KUKA KRL program: gestion_camara.src, gestion_camara.dat

--- gestion_camara.src ---
&ACCESS RVO2
&REL 8
&PARAM EDITMASK = *
&PARAM TEMPLATE = C:\KRC\Roboter\Template\vorgabe
DEF gestion_camara( )


END
GLOBAL DEF CAM_INI()

INPICKER_Handler.DataToSend.command=0
INPICKER_Handler.DataToSend.CameraID=0
INPICKER_Handler.DataToSend.ContainerID=0
INPICKER_Handler.DataToSend.GraspConfirmation=0
INPICKER_Handler.datatosend.partid=0

END
GLOBAL DEF CAM_CALIB_INI()

INPICKER_Handler.DataToSend.command=0
INPICKER_Handler.DataToSend.CameraID=1
INPICKER_Handler.DataToSend.ContainerID=0
INPICKER_Handler.DataToSend.GraspConfirmation=0
INPICKER_Handler.datatosend.partid=1

END

GLOBAL DEF CAM_CALIB_FOTO(P_IN :IN)
INT P_IN

INPICKER_Handler.DataToSend.command=0
wait for (INPICKER_Handler.DataReceived.state==0)
INPICKER_Handler.DataToSend.GraspConfirmation=P_IN
INPICKER_Handler.DataToSend.command=3
wait for (INPICKER_Handler.DataReceived.state==30)

END

GLOBAL DEF CAM_CALIB_END()


INPICKER_Handler.DataToSend.command=0
wait for (INPICKER_Handler.DataReceived.state==0)
INPICKER_Handler.DataToSend.command=4
wait for (INPICKER_Handler.DataReceived.state==30)

END

--- gestion_camara.dat ---
&ACCESS RVO2
&REL 8
&PARAM EDITMASK = *
&PARAM TEMPLATE = C:\KRC\Roboter\Template\vorgabe
DEFDAT gestion_camara
;FOLD EXTERNAL DECLARATIONS;%{PE}%MKUKATPBASIS,%CEXT,%VCOMMON,%P
;FOLD GRIPPERTECH EXT
  EXT  H50 (INT:IN, INT:IN ,INT:IN ,GRP_TYP:IN)
;ENDFOLD (GRIPPERTECH EXT)
;FOLD SPOTTECH EXT
  EXT  USERSPOT (S_COMMAND  :IN, SPOT_TYPE:IN)
;ENDFOLD (SPOTTECH EXT)
;FOLD BASISTECH EXT;%{PE}%MKUKATPBASIS,%CEXT,%VEXT,%P
EXT  BAS (BAS_COMMAND  :IN,REAL  :IN )
DECL INT SUCCESS
;ENDFOLD (BASISTECH EXT)
;FOLD USER EXT;%{E}%MKUKATPUSER,%CEXT,%VEXT,%P
;Make your modifications here

;ENDFOLD (USER EXT)
;ENDFOLD (EXTERNAL DECLARATIONS)
ENDDAT
